// TIA Portal V20 export
ORGANIZATION_BLOCK "Startup_1"   // OB100, LAD, Startup
TITLE = "Complete Restart"
{ S7_Optimized_Access := 'TRUE' }
// stored: SetENOAutomatically false
   VAR_INPUT
      LostRetentive : Bool;   // True if retentive data are lost
      LostRTC : Bool;   // True if date and time are lost
   END_VAR
   VAR_TEMP
      NumberOf_Reset : Int;
   END_VAR
BEGIN

REGION Network 1
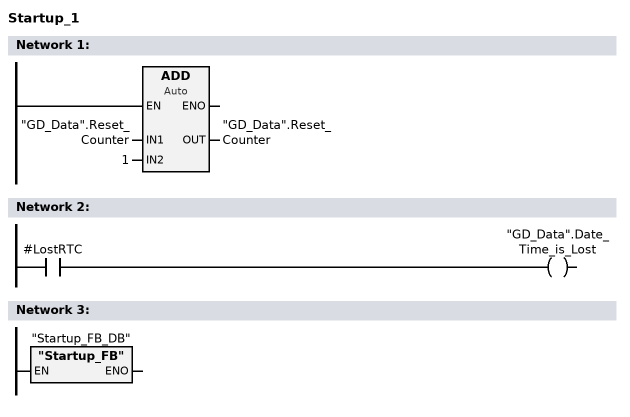
   RUNG wire#powerrail
      { S7_GenerateENO := "TRUE" } Add(in1 := "GD_Data".Reset_Counter, in2 := 1, out => "GD_Data".Reset_Counter)
   END_RUNG
   // the same network as SCL:
   "GD_Data".Reset_Counter := "GD_Data".Reset_Counter + 1;
END_REGION

REGION Network 2
   RUNG wire#powerrail
      Contact( #LostRTC )
      Coil( "GD_Data".Date_Time_is_Lost )
   END_RUNG
   // the same network as SCL:
   "GD_Data".Date_Time_is_Lost := #LostRTC;
END_REGION

REGION Network 3
   RUNG wire#powerrail
      "Startup_FB_DB"()
   END_RUNG
   // the same network as SCL:
   "Startup_FB_DB"();   // "Startup_FB"
END_REGION
END_ORGANIZATION_BLOCK
